PROGRAM F02_METS_DoubleInputs

VAR
	fbLiftComplete					: FB_IO2_DoubleInputCtrl;	(*ib61KF1_6_StackLifted_SFWM and ib62KF1_3_StackLiftedSensor*)
	fbStackComplete				: FB_IO2_DoubleInputCtrl;	(*ib61KF1_2_StackComplete_SFWM and ib62KF1_7_StackCompletedSensor*)
	fbBundleCrossPushComplete		: FB_IO2_DoubleInputCtrl;	(*ib61KF1_7_BundleCrossPush_SFWM and ib62KF1_4_BundleCrossPushSensor*)
	fbBundleTranferComplete		: FB_IO2_DoubleInputCtrl;	(*ib61KF1_4_BundleTransferComplete_SFWM and ib62KF1_8_BundleTranferCompleteSensor*)

	fbRowComplete				: FB_IO2_DoubleInputCtrl;	(*ib161KF1_3_RowComplete_SFCP and ib163KF1_2_RowCompleteSensor*)
	fbLayerComplete				: FB_IO2_DoubleInputCtrl;	(*ib161KF1_7_LayerComplete_SFCP and ib163KF1_6_LayerCompleteSensor*)
	fbCaseComplete				: FB_IO2_DoubleInputCtrl;	(*ib161KF1_4_CaseComplete_SFCP and ib163KF1_3_CaseCompleteSensor*)
	fbCaseDischarge				: FB_IO2_DoubleInputCtrl;	(*ib161KF1_8_CaseDischarged_SFCP and ib163KF1_7_CaseDischargedSensor*)
	fbCaseLabelValidationTrigSensor	: FB_IO2_DoubleInputCtrl;	(* and *)
	fbIntermediatePush				: FB_IO2_DoubleInputCtrl;	(* and *)

	fbCaseArrived					: FB_IO2_DoubleInputCtrl;
	fbCaseTransit					: FB_IO2_DoubleInputCtrl;
	fbCasePlaced					: FB_IO2_DoubleInputCtrl;
	fbPalletCompleted				: FB_IO2_DoubleInputCtrl;

	tonSettingsValideDelay			: TON;

	fbRowCompleteSensorCTU		: FB_CTU32;	(*RowComplete*)
	fbRowCompleteMachineCTU		: FB_CTU32;
	fbRowCompleteCTU				: FB_CTU32;

	fbLayerCompleteSensorCTU		: FB_CTU32;	(*LayerComplete*)
	fbLayerCompleteMachineCTU		: FB_CTU32;
	fbLayerCompleteCTU			: FB_CTU32;

	fbCaseCompleteSensorCTU		: FB_CTU32;	(*CaseComplete*)
	fbCaseCompleteMachineCTU		: FB_CTU32;
	fbCaseCompleteCTU				: FB_CTU32;

	fbCaseDischargedSensorCTU		: FB_CTU32;	(*CaseDischarged*)
	fbCaseDischargedMachineCTU		: FB_CTU32;
	fbCaseDischargedCTU			: FB_CTU32;

	fbCaseLabelValidationSensorCTU	: FB_CTU32;	(*CaseLabelValidation*)
	fbCaseLabelValidationMachineCTU	: FB_CTU32;
	fbCaseLabelValidationCTU		: FB_CTU32;

END_VAR


(*
Modification history:
Date		|	Author 		|	Remark
----------------------------------------------------------------------------------------------------
16.09.20	|	PP			|	Start Remarking.
*)

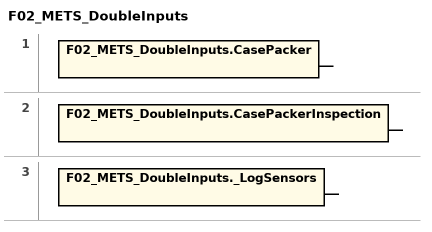
// NETWORK 1
F02_METS_DoubleInputs.CasePacker();

// NETWORK 2
F02_METS_DoubleInputs.CasePackerInspection();

// NETWORK 3
F02_METS_DoubleInputs._LogSensors();

ACTION _LogSensors:
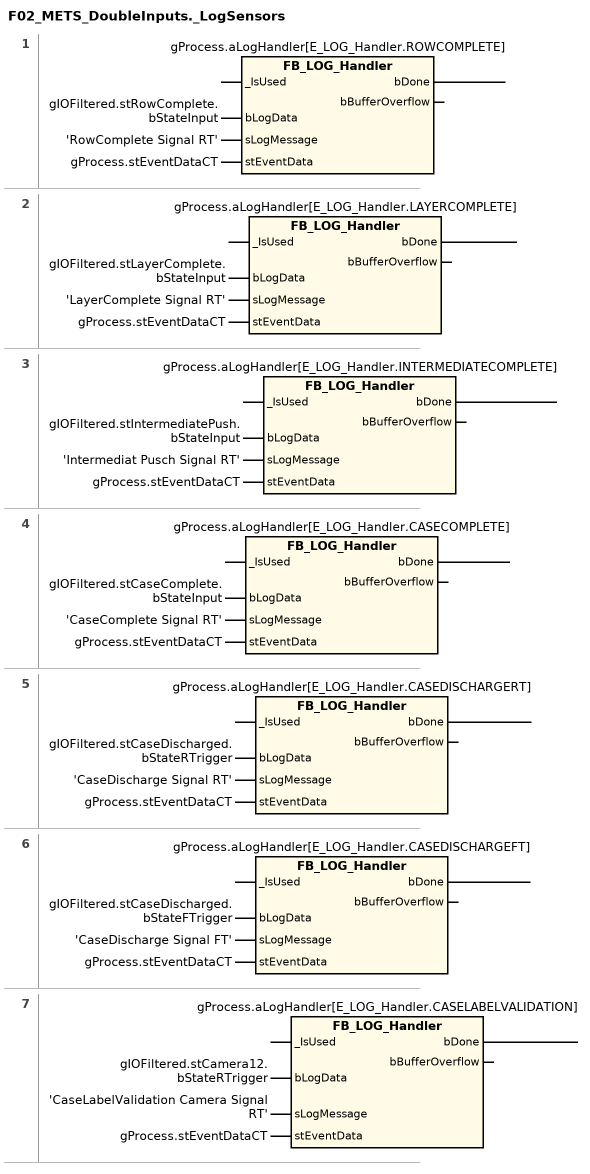
// NETWORK 1
gProcess.aLogHandler[E_LOG_Handler.ROWCOMPLETE](
    bLogData := gIOFiltered.stRowComplete.bStateInput,
    sLogMessage := 'RowComplete Signal RT',
    stEventData := gProcess.stEventDataCT); // FB_LOG_Handler

// NETWORK 2
gProcess.aLogHandler[E_LOG_Handler.LAYERCOMPLETE](
    bLogData := gIOFiltered.stLayerComplete.bStateInput,
    sLogMessage := 'LayerComplete Signal RT',
    stEventData := gProcess.stEventDataCT); // FB_LOG_Handler

// NETWORK 3
gProcess.aLogHandler[E_LOG_Handler.INTERMEDIATECOMPLETE](
    bLogData := gIOFiltered.stIntermediatePush.bStateInput,
    sLogMessage := 'Intermediat Pusch Signal RT',
    stEventData := gProcess.stEventDataCT); // FB_LOG_Handler

// NETWORK 4
gProcess.aLogHandler[E_LOG_Handler.CASECOMPLETE](
    bLogData := gIOFiltered.stCaseComplete.bStateInput,
    sLogMessage := 'CaseComplete Signal RT',
    stEventData := gProcess.stEventDataCT); // FB_LOG_Handler

// NETWORK 5
gProcess.aLogHandler[E_LOG_Handler.CASEDISCHARGERT](
    bLogData := gIOFiltered.stCaseDischarged.bStateRTrigger,
    sLogMessage := 'CaseDischarge Signal RT',
    stEventData := gProcess.stEventDataCT); // FB_LOG_Handler

// NETWORK 6
gProcess.aLogHandler[E_LOG_Handler.CASEDISCHARGEFT](
    bLogData := gIOFiltered.stCaseDischarged.bStateFTrigger,
    sLogMessage := 'CaseDischarge Signal FT',
    stEventData := gProcess.stEventDataCT); // FB_LOG_Handler

// NETWORK 7
gProcess.aLogHandler[E_LOG_Handler.CASELABELVALIDATION](
    bLogData := gIOFiltered.stCamera12.bStateRTrigger,
    sLogMessage := 'CaseLabelValidation Camera Signal RT',
    stEventData := gProcess.stEventDataCT); // FB_LOG_Handler
END_ACTION

ACTION CasePacker:
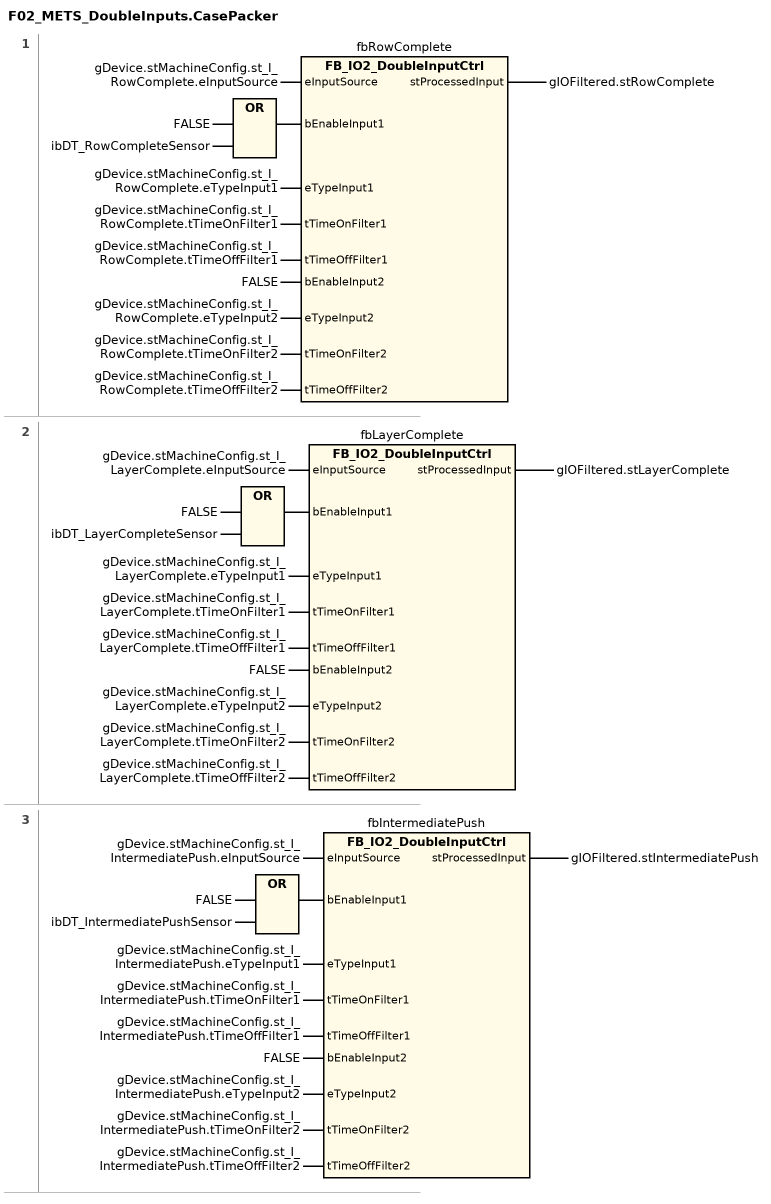
// NETWORK 1
fbRowComplete(
    eInputSource := gDevice.stMachineConfig.st_I_RowComplete.eInputSource,
    bEnableInput1 := FALSE OR ibDT_RowCompleteSensor,
    eTypeInput1 := gDevice.stMachineConfig.st_I_RowComplete.eTypeInput1,
    tTimeOnFilter1 := gDevice.stMachineConfig.st_I_RowComplete.tTimeOnFilter1,
    tTimeOffFilter1 := gDevice.stMachineConfig.st_I_RowComplete.tTimeOffFilter1,
    bEnableInput2 := FALSE,
    eTypeInput2 := gDevice.stMachineConfig.st_I_RowComplete.eTypeInput2,
    tTimeOnFilter2 := gDevice.stMachineConfig.st_I_RowComplete.tTimeOnFilter2,
    tTimeOffFilter2 := gDevice.stMachineConfig.st_I_RowComplete.tTimeOffFilter2); // FB_IO2_DoubleInputCtrl
gIOFiltered.stRowComplete := fbRowComplete.stProcessedInput;

// NETWORK 2
fbLayerComplete(
    eInputSource := gDevice.stMachineConfig.st_I_LayerComplete.eInputSource,
    bEnableInput1 := FALSE OR ibDT_LayerCompleteSensor,
    eTypeInput1 := gDevice.stMachineConfig.st_I_LayerComplete.eTypeInput1,
    tTimeOnFilter1 := gDevice.stMachineConfig.st_I_LayerComplete.tTimeOnFilter1,
    tTimeOffFilter1 := gDevice.stMachineConfig.st_I_LayerComplete.tTimeOffFilter1,
    bEnableInput2 := FALSE,
    eTypeInput2 := gDevice.stMachineConfig.st_I_LayerComplete.eTypeInput2,
    tTimeOnFilter2 := gDevice.stMachineConfig.st_I_LayerComplete.tTimeOnFilter2,
    tTimeOffFilter2 := gDevice.stMachineConfig.st_I_LayerComplete.tTimeOffFilter2); // FB_IO2_DoubleInputCtrl
gIOFiltered.stLayerComplete := fbLayerComplete.stProcessedInput;

// NETWORK 3
fbIntermediatePush(
    eInputSource := gDevice.stMachineConfig.st_I_IntermediatePush.eInputSource,
    bEnableInput1 := FALSE OR ibDT_IntermediatePushSensor,
    eTypeInput1 := gDevice.stMachineConfig.st_I_IntermediatePush.eTypeInput1,
    tTimeOnFilter1 := gDevice.stMachineConfig.st_I_IntermediatePush.tTimeOnFilter1,
    tTimeOffFilter1 := gDevice.stMachineConfig.st_I_IntermediatePush.tTimeOffFilter1,
    bEnableInput2 := FALSE,
    eTypeInput2 := gDevice.stMachineConfig.st_I_IntermediatePush.eTypeInput2,
    tTimeOnFilter2 := gDevice.stMachineConfig.st_I_IntermediatePush.tTimeOnFilter2,
    tTimeOffFilter2 := gDevice.stMachineConfig.st_I_IntermediatePush.tTimeOffFilter2); // FB_IO2_DoubleInputCtrl
gIOFiltered.stIntermediatePush := fbIntermediatePush.stProcessedInput;

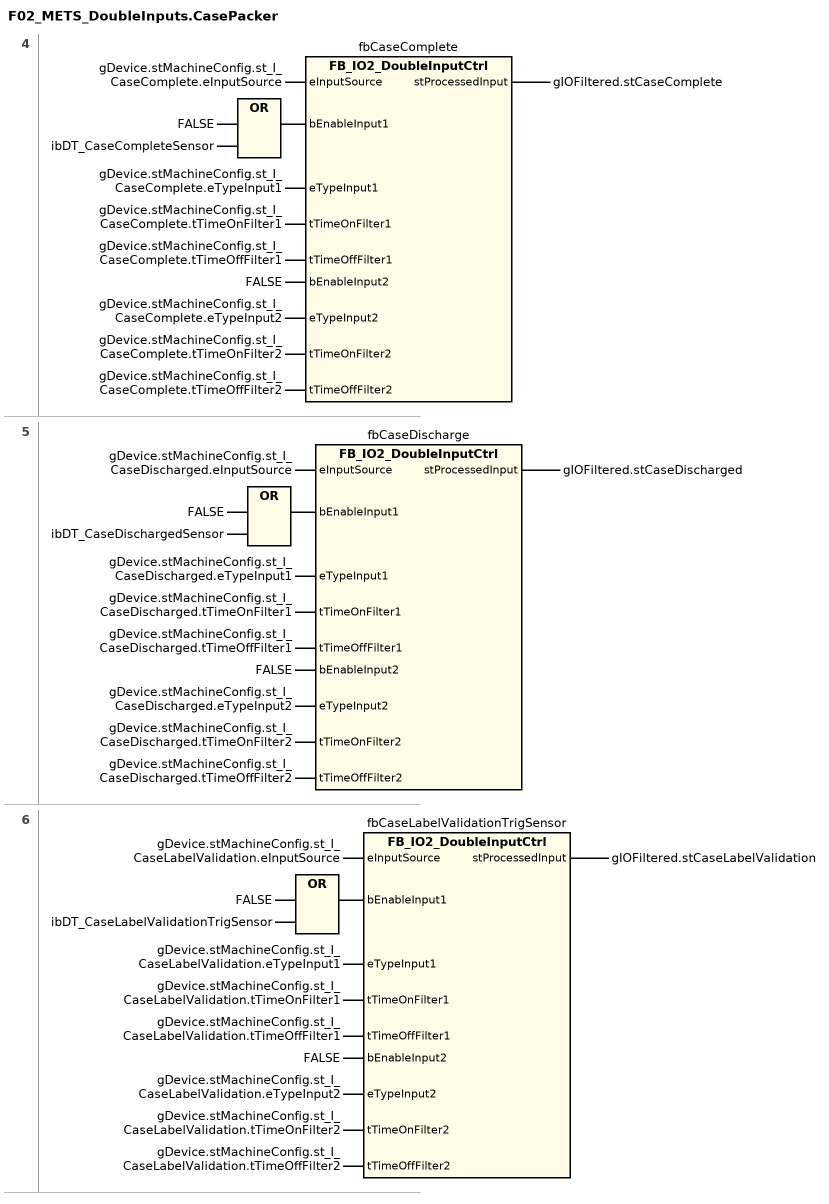
// NETWORK 4
fbCaseComplete(
    eInputSource := gDevice.stMachineConfig.st_I_CaseComplete.eInputSource,
    bEnableInput1 := FALSE OR ibDT_CaseCompleteSensor,
    eTypeInput1 := gDevice.stMachineConfig.st_I_CaseComplete.eTypeInput1,
    tTimeOnFilter1 := gDevice.stMachineConfig.st_I_CaseComplete.tTimeOnFilter1,
    tTimeOffFilter1 := gDevice.stMachineConfig.st_I_CaseComplete.tTimeOffFilter1,
    bEnableInput2 := FALSE,
    eTypeInput2 := gDevice.stMachineConfig.st_I_CaseComplete.eTypeInput2,
    tTimeOnFilter2 := gDevice.stMachineConfig.st_I_CaseComplete.tTimeOnFilter2,
    tTimeOffFilter2 := gDevice.stMachineConfig.st_I_CaseComplete.tTimeOffFilter2); // FB_IO2_DoubleInputCtrl
gIOFiltered.stCaseComplete := fbCaseComplete.stProcessedInput;

// NETWORK 5
fbCaseDischarge(
    eInputSource := gDevice.stMachineConfig.st_I_CaseDischarged.eInputSource,
    bEnableInput1 := FALSE OR ibDT_CaseDischargedSensor,
    eTypeInput1 := gDevice.stMachineConfig.st_I_CaseDischarged.eTypeInput1,
    tTimeOnFilter1 := gDevice.stMachineConfig.st_I_CaseDischarged.tTimeOnFilter1,
    tTimeOffFilter1 := gDevice.stMachineConfig.st_I_CaseDischarged.tTimeOffFilter1,
    bEnableInput2 := FALSE,
    eTypeInput2 := gDevice.stMachineConfig.st_I_CaseDischarged.eTypeInput2,
    tTimeOnFilter2 := gDevice.stMachineConfig.st_I_CaseDischarged.tTimeOnFilter2,
    tTimeOffFilter2 := gDevice.stMachineConfig.st_I_CaseDischarged.tTimeOffFilter2); // FB_IO2_DoubleInputCtrl
gIOFiltered.stCaseDischarged := fbCaseDischarge.stProcessedInput;

// NETWORK 6
fbCaseLabelValidationTrigSensor(
    eInputSource := gDevice.stMachineConfig.st_I_CaseLabelValidation.eInputSource,
    bEnableInput1 := FALSE OR ibDT_CaseLabelValidationTrigSensor,
    eTypeInput1 := gDevice.stMachineConfig.st_I_CaseLabelValidation.eTypeInput1,
    tTimeOnFilter1 := gDevice.stMachineConfig.st_I_CaseLabelValidation.tTimeOnFilter1,
    tTimeOffFilter1 := gDevice.stMachineConfig.st_I_CaseLabelValidation.tTimeOffFilter1,
    bEnableInput2 := FALSE,
    eTypeInput2 := gDevice.stMachineConfig.st_I_CaseLabelValidation.eTypeInput2,
    tTimeOnFilter2 := gDevice.stMachineConfig.st_I_CaseLabelValidation.tTimeOnFilter2,
    tTimeOffFilter2 := gDevice.stMachineConfig.st_I_CaseLabelValidation.tTimeOffFilter2); // FB_IO2_DoubleInputCtrl
gIOFiltered.stCaseLabelValidation := fbCaseLabelValidationTrigSensor.stProcessedInput;
END_ACTION

ACTION CasePackerInspection:
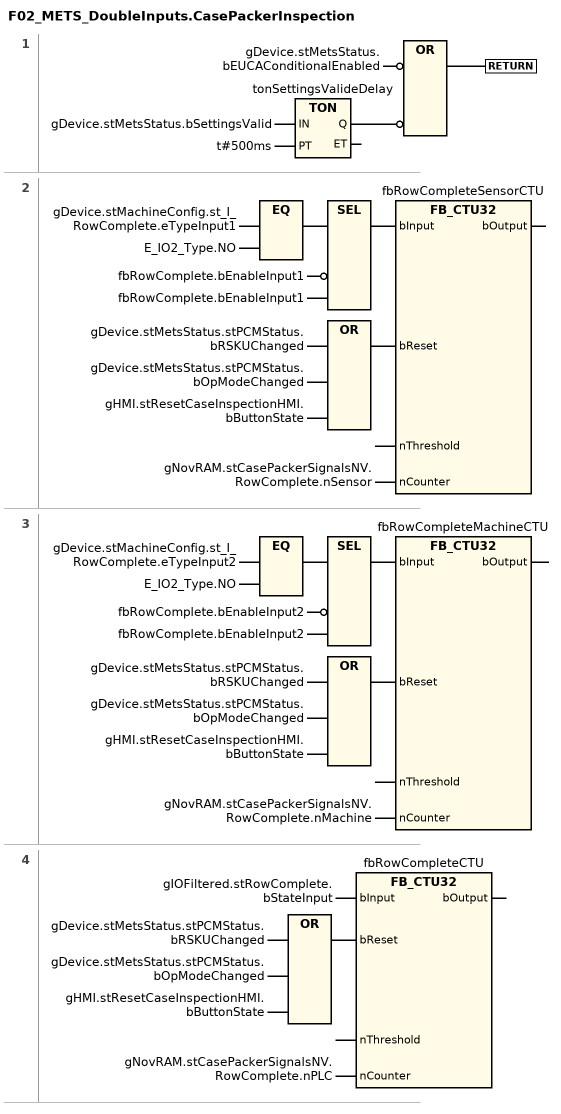
// NETWORK 1
tonSettingsValideDelay(IN := gDevice.stMetsStatus.bSettingsValid, PT := t#500ms); // TON
IF NOT gDevice.stMetsStatus.bEUCAConditionalEnabled OR NOT tonSettingsValideDelay.Q THEN RETURN; END_IF

// NETWORK 2
fbRowCompleteSensorCTU(
    bInput := SEL(gDevice.stMachineConfig.st_I_RowComplete.eTypeInput1 = E_IO2_Type.NO, NOT fbRowComplete.bEnableInput1, fbRowComplete.bEnableInput1),
    bReset := gDevice.stMetsStatus.stPCMStatus.bRSKUChanged OR gDevice.stMetsStatus.stPCMStatus.bOpModeChanged OR gHMI.stResetCaseInspectionHMI.bButtonState,
    nCounter := gNovRAM.stCasePackerSignalsNV.RowComplete.nSensor); // FB_CTU32

// NETWORK 3
fbRowCompleteMachineCTU(
    bInput := SEL(gDevice.stMachineConfig.st_I_RowComplete.eTypeInput2 = E_IO2_Type.NO, NOT fbRowComplete.bEnableInput2, fbRowComplete.bEnableInput2),
    bReset := gDevice.stMetsStatus.stPCMStatus.bRSKUChanged OR gDevice.stMetsStatus.stPCMStatus.bOpModeChanged OR gHMI.stResetCaseInspectionHMI.bButtonState,
    nCounter := gNovRAM.stCasePackerSignalsNV.RowComplete.nMachine); // FB_CTU32

// NETWORK 4
fbRowCompleteCTU(
    bInput := gIOFiltered.stRowComplete.bStateInput,
    bReset := gDevice.stMetsStatus.stPCMStatus.bRSKUChanged OR gDevice.stMetsStatus.stPCMStatus.bOpModeChanged OR gHMI.stResetCaseInspectionHMI.bButtonState,
    nCounter := gNovRAM.stCasePackerSignalsNV.RowComplete.nPLC); // FB_CTU32

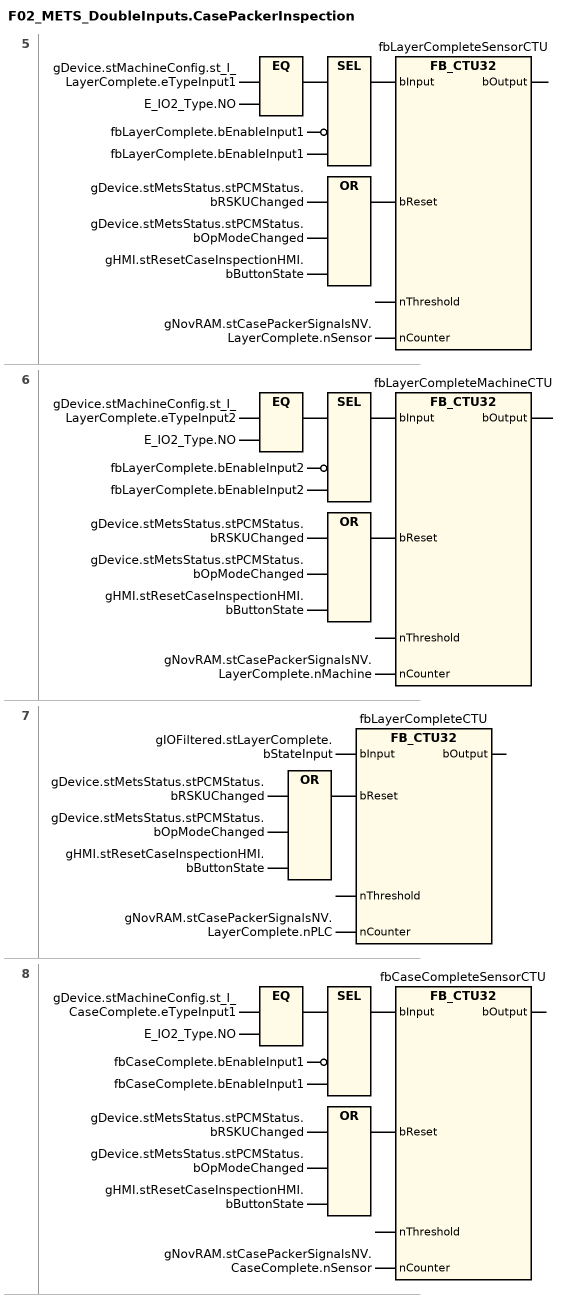
// NETWORK 5
fbLayerCompleteSensorCTU(
    bInput := SEL(gDevice.stMachineConfig.st_I_LayerComplete.eTypeInput1 = E_IO2_Type.NO, NOT fbLayerComplete.bEnableInput1, fbLayerComplete.bEnableInput1),
    bReset := gDevice.stMetsStatus.stPCMStatus.bRSKUChanged OR gDevice.stMetsStatus.stPCMStatus.bOpModeChanged OR gHMI.stResetCaseInspectionHMI.bButtonState,
    nCounter := gNovRAM.stCasePackerSignalsNV.LayerComplete.nSensor); // FB_CTU32

// NETWORK 6
fbLayerCompleteMachineCTU(
    bInput := SEL(gDevice.stMachineConfig.st_I_LayerComplete.eTypeInput2 = E_IO2_Type.NO, NOT fbLayerComplete.bEnableInput2, fbLayerComplete.bEnableInput2),
    bReset := gDevice.stMetsStatus.stPCMStatus.bRSKUChanged OR gDevice.stMetsStatus.stPCMStatus.bOpModeChanged OR gHMI.stResetCaseInspectionHMI.bButtonState,
    nCounter := gNovRAM.stCasePackerSignalsNV.LayerComplete.nMachine); // FB_CTU32

// NETWORK 7
fbLayerCompleteCTU(
    bInput := gIOFiltered.stLayerComplete.bStateInput,
    bReset := gDevice.stMetsStatus.stPCMStatus.bRSKUChanged OR gDevice.stMetsStatus.stPCMStatus.bOpModeChanged OR gHMI.stResetCaseInspectionHMI.bButtonState,
    nCounter := gNovRAM.stCasePackerSignalsNV.LayerComplete.nPLC); // FB_CTU32

// NETWORK 8
fbCaseCompleteSensorCTU(
    bInput := SEL(gDevice.stMachineConfig.st_I_CaseComplete.eTypeInput1 = E_IO2_Type.NO, NOT fbCaseComplete.bEnableInput1, fbCaseComplete.bEnableInput1),
    bReset := gDevice.stMetsStatus.stPCMStatus.bRSKUChanged OR gDevice.stMetsStatus.stPCMStatus.bOpModeChanged OR gHMI.stResetCaseInspectionHMI.bButtonState,
    nCounter := gNovRAM.stCasePackerSignalsNV.CaseComplete.nSensor); // FB_CTU32

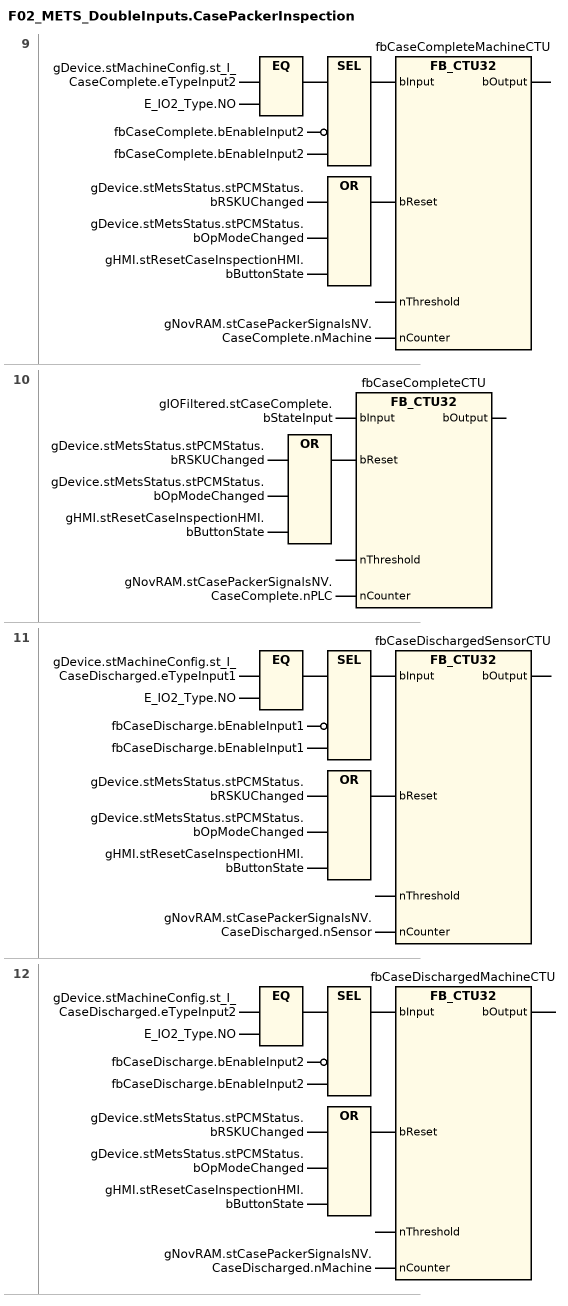
// NETWORK 9
fbCaseCompleteMachineCTU(
    bInput := SEL(gDevice.stMachineConfig.st_I_CaseComplete.eTypeInput2 = E_IO2_Type.NO, NOT fbCaseComplete.bEnableInput2, fbCaseComplete.bEnableInput2),
    bReset := gDevice.stMetsStatus.stPCMStatus.bRSKUChanged OR gDevice.stMetsStatus.stPCMStatus.bOpModeChanged OR gHMI.stResetCaseInspectionHMI.bButtonState,
    nCounter := gNovRAM.stCasePackerSignalsNV.CaseComplete.nMachine); // FB_CTU32

// NETWORK 10
fbCaseCompleteCTU(
    bInput := gIOFiltered.stCaseComplete.bStateInput,
    bReset := gDevice.stMetsStatus.stPCMStatus.bRSKUChanged OR gDevice.stMetsStatus.stPCMStatus.bOpModeChanged OR gHMI.stResetCaseInspectionHMI.bButtonState,
    nCounter := gNovRAM.stCasePackerSignalsNV.CaseComplete.nPLC); // FB_CTU32

// NETWORK 11
fbCaseDischargedSensorCTU(
    bInput := SEL(gDevice.stMachineConfig.st_I_CaseDischarged.eTypeInput1 = E_IO2_Type.NO, NOT fbCaseDischarge.bEnableInput1, fbCaseDischarge.bEnableInput1),
    bReset := gDevice.stMetsStatus.stPCMStatus.bRSKUChanged OR gDevice.stMetsStatus.stPCMStatus.bOpModeChanged OR gHMI.stResetCaseInspectionHMI.bButtonState,
    nCounter := gNovRAM.stCasePackerSignalsNV.CaseDischarged.nSensor); // FB_CTU32

// NETWORK 12
fbCaseDischargedMachineCTU(
    bInput := SEL(gDevice.stMachineConfig.st_I_CaseDischarged.eTypeInput2 = E_IO2_Type.NO, NOT fbCaseDischarge.bEnableInput2, fbCaseDischarge.bEnableInput2),
    bReset := gDevice.stMetsStatus.stPCMStatus.bRSKUChanged OR gDevice.stMetsStatus.stPCMStatus.bOpModeChanged OR gHMI.stResetCaseInspectionHMI.bButtonState,
    nCounter := gNovRAM.stCasePackerSignalsNV.CaseDischarged.nMachine); // FB_CTU32

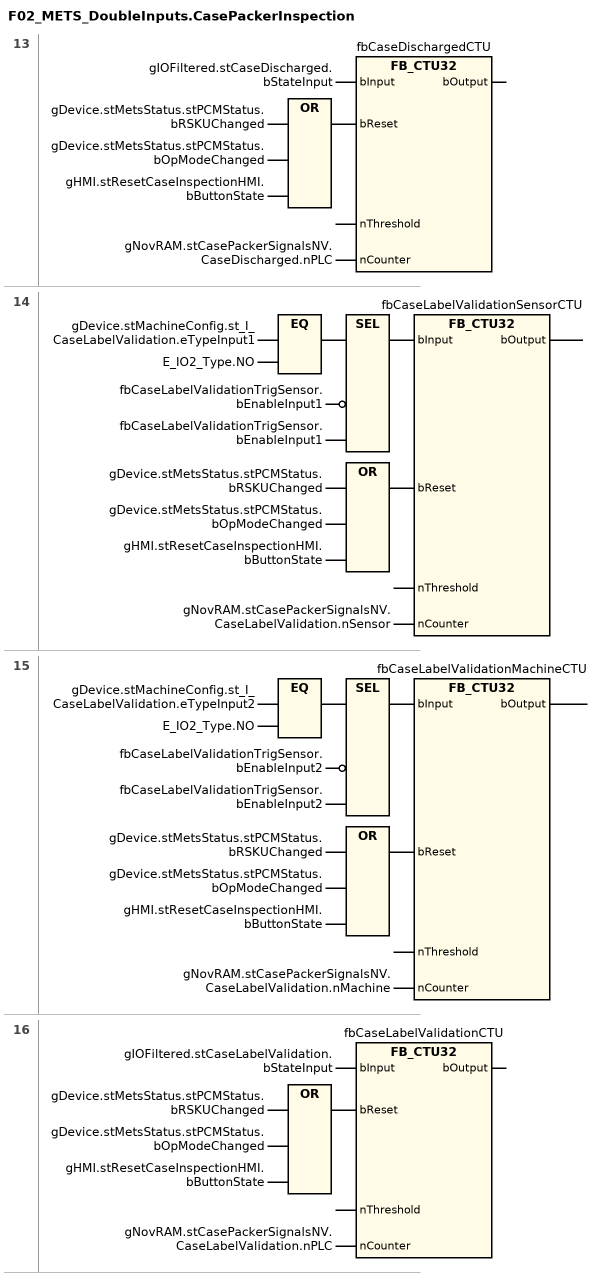
// NETWORK 13
fbCaseDischargedCTU(
    bInput := gIOFiltered.stCaseDischarged.bStateInput,
    bReset := gDevice.stMetsStatus.stPCMStatus.bRSKUChanged OR gDevice.stMetsStatus.stPCMStatus.bOpModeChanged OR gHMI.stResetCaseInspectionHMI.bButtonState,
    nCounter := gNovRAM.stCasePackerSignalsNV.CaseDischarged.nPLC); // FB_CTU32

// NETWORK 14
fbCaseLabelValidationSensorCTU(
    bInput := SEL(gDevice.stMachineConfig.st_I_CaseLabelValidation.eTypeInput1 = E_IO2_Type.NO, NOT fbCaseLabelValidationTrigSensor.bEnableInput1, fbCaseLabelValidationTrigSensor.bEnableInput1),
    bReset := gDevice.stMetsStatus.stPCMStatus.bRSKUChanged OR gDevice.stMetsStatus.stPCMStatus.bOpModeChanged OR gHMI.stResetCaseInspectionHMI.bButtonState,
    nCounter := gNovRAM.stCasePackerSignalsNV.CaseLabelValidation.nSensor); // FB_CTU32

// NETWORK 15
fbCaseLabelValidationMachineCTU(
    bInput := SEL(gDevice.stMachineConfig.st_I_CaseLabelValidation.eTypeInput2 = E_IO2_Type.NO, NOT fbCaseLabelValidationTrigSensor.bEnableInput2, fbCaseLabelValidationTrigSensor.bEnableInput2),
    bReset := gDevice.stMetsStatus.stPCMStatus.bRSKUChanged OR gDevice.stMetsStatus.stPCMStatus.bOpModeChanged OR gHMI.stResetCaseInspectionHMI.bButtonState,
    nCounter := gNovRAM.stCasePackerSignalsNV.CaseLabelValidation.nMachine); // FB_CTU32

// NETWORK 16
fbCaseLabelValidationCTU(
    bInput := gIOFiltered.stCaseLabelValidation.bStateInput,
    bReset := gDevice.stMetsStatus.stPCMStatus.bRSKUChanged OR gDevice.stMetsStatus.stPCMStatus.bOpModeChanged OR gHMI.stResetCaseInspectionHMI.bButtonState,
    nCounter := gNovRAM.stCasePackerSignalsNV.CaseLabelValidation.nPLC); // FB_CTU32
END_ACTION

END_PROGRAM

(* stored: Version 1.1.0.1
   POU F02_METS_DoubleInputs: Id {8386c294-eb97-4d8f-8031-bf34b8a3f1c7}, SpecialFunc None
   Action _LogSensors: Id {5735df9c-aae8-4194-aba9-515a980deee7}
   Action CasePacker: Id {a8b7de69-ab91-428f-a01a-d7d18a31ea5f}
   Action CasePackerInspection: Id {3b4b7b23-b88a-45ed-b885-b1123a89ad4d} *)
